TYPE T_Position : DINT; END_TYPE

(* stored: Version 1.1.0.1, ProductVersion 3.1.4024.4
   DUT T_Position: Id {afd84c02-4bca-432a-abd9-9aca660f6c08} *)
